(* IEC 61131-3 sources: verifaps-lib/share/PPU.stold (part 7) *)

    Pusher_states_t#PusherY1_Move_Out_White:
        {* begin(State) *}
        {* begin(onEntry) *}
        _transit := FALSE;
        {* end(onEntry) *}
        {* begin(onActive) *}
        IF ((SorterPusher1MovedOut = FALSE) AND (SorterPusher1MovedIn = TRUE)) THEN
            PusherY1 := TRUE;
        END_IF;
        {* end(onActive) *}
        {* begin(transition) *}
        IF SorterPusher1MovedOut THEN
            _transit := TRUE;
            _state := Pusher_states_t#Wait_Y1_White;
        END_IF;
        {* end(transition) *}
        {* begin(onExit) *}
        {* end(onExit) *}
        {* end(State) *}

    Pusher_states_t#PusherY2_Move_In_Black:
        {* begin(State) *}
        {* begin(onEntry) *}
        _transit := FALSE;
        {* end(onEntry) *}
        {* begin(onActive) *}
        IF ((SorterPusher2MovedOut = TRUE) AND (SorterPusher2MovedIn = FALSE)) THEN
            PusherY2 := FALSE;
        END_IF;
        {* end(onActive) *}
        {* begin(transition) *}
        IF SorterPusher2MovedIn THEN
            _transit := TRUE;
            _state := Pusher_states_t#Reset_interconnect_Slide2_Black;
        END_IF;
        {* end(transition) *}
        {* begin(onExit) *}
        {* end(onExit) *}
        {* end(State) *}

    Pusher_states_t#PusherY2_Move_In_Metal:
        {* begin(State) *}
        {* begin(onEntry) *}
        _transit := FALSE;
        {* end(onEntry) *}
        {* begin(onActive) *}
        IF ((SorterPusher2MovedOut = TRUE) AND (SorterPusher2MovedIn = FALSE)) THEN
            PusherY2 := FALSE;
        END_IF;
        {* end(onActive) *}
        {* begin(transition) *}
        IF SorterPusher2MovedIn THEN
            _transit := TRUE;
            _state := Pusher_states_t#Reset_interconnect_Slide2_Metal;
        END_IF;
        {* end(transition) *}
        {* begin(onExit) *}
        {* end(onExit) *}
        {* end(State) *}

    Pusher_states_t#PusherY2_Move_In_White:
        {* begin(State) *}
        {* begin(onEntry) *}
        _transit := FALSE;
        {* end(onEntry) *}
        {* begin(onActive) *}
        IF ((SorterPusher2MovedOut = TRUE) AND (SorterPusher2MovedIn = FALSE)) THEN
            PusherY2 := FALSE;
        END_IF;
        {* end(onActive) *}
        {* begin(transition) *}
        IF SorterPusher2MovedIn THEN
            _transit := TRUE;
            _state := Pusher_states_t#Reset_interconnect_Slide2_White;
        END_IF;
        {* end(transition) *}
        {* begin(onExit) *}
        {* end(onExit) *}
        {* end(State) *}

    Pusher_states_t#PusherY2_Move_Out_Black:
        {* begin(State) *}
        {* begin(onEntry) *}
        _transit := FALSE;
        {* end(onEntry) *}
        {* begin(onActive) *}
        IF ((SorterPusher2MovedOut = FALSE) AND (SorterPusher2MovedIn = TRUE)) THEN
            PusherY2 := TRUE;
        END_IF;
        {* end(onActive) *}
        {* begin(transition) *}
        IF SorterPusher2MovedOut THEN
            _transit := TRUE;
            _state := Pusher_states_t#Wait_Y2_Black;
        END_IF;
        {* end(transition) *}
        {* begin(onExit) *}
        {* end(onExit) *}
        {* end(State) *}

    Pusher_states_t#PusherY2_Move_Out_Metal:
        {* begin(State) *}
        {* begin(onEntry) *}
        _transit := FALSE;
        {* end(onEntry) *}
        {* begin(onActive) *}
        IF ((SorterPusher2MovedOut = FALSE) AND (SorterPusher2MovedIn = TRUE)) THEN
            PusherY2 := TRUE;
        END_IF;
        {* end(onActive) *}
        {* begin(transition) *}
        IF SorterPusher2MovedOut THEN
            _transit := TRUE;
            _state := Pusher_states_t#Wait_Y2_Metal;
        END_IF;
        {* end(transition) *}
        {* begin(onExit) *}
        {* end(onExit) *}
        {* end(State) *}

    Pusher_states_t#PusherY2_Move_Out_White:
        {* begin(State) *}
        {* begin(onEntry) *}
        _transit := FALSE;
        {* end(onEntry) *}
        {* begin(onActive) *}
        IF ((SorterPusher2MovedOut = FALSE) AND (SorterPusher2MovedIn = TRUE)) THEN
            PusherY2 := TRUE;
        END_IF;
        {* end(onActive) *}
        {* begin(transition) *}
        IF SorterPusher2MovedOut THEN
            _transit := TRUE;
            _state := Pusher_states_t#Wait_Y2_White;
        END_IF;
        {* end(transition) *}
        {* begin(onExit) *}
        {* end(onExit) *}
        {* end(State) *}

    Pusher_states_t#Reset_interconnect3:
        {* begin(State) *}
        {* begin(onEntry) *}
        _transit := FALSE;
        {* end(onEntry) *}
        {* begin(onActive) *}
        interconnect2 := FALSE;
        Timer2(IN := FALSE, PT := TIME#);
        Slide3_black := (Slide3_black - INT#1);
        Priority_Var_Black := (Priority_Var_Black - INT#1);
        {* end(onActive) *}
        {* begin(transition) *}
        IF TRUE THEN
            _transit := TRUE;
            _state := Pusher_states_t#Interstep_2;
        END_IF;
        {* end(transition) *}
        {* begin(onExit) *}
        {* end(onExit) *}
        {* end(State) *}

    Pusher_states_t#Reset_interconnect_Slide1_Black:
        {* begin(State) *}
        {* begin(onEntry) *}
        _transit := FALSE;
        {* end(onEntry) *}
        {* begin(onActive) *}
        interconnect3 := FALSE;
        Timer3(IN := FALSE, PT := TIME#);
        interconnect_Slide1_Black := FALSE;
        Timer_Slide1_Black(IN := FALSE, PT := TIME#);
        Slide1_black := (Slide1_black - INT#1);
        Priority_Var_Black := (Priority_Var_Black - INT#1);
        {* end(onActive) *}
        {* begin(transition) *}
        IF TRUE THEN
            _transit := TRUE;
            _state := Pusher_states_t#Interstep_2;
        END_IF;
        {* end(transition) *}
        {* begin(onExit) *}
        {* end(onExit) *}
        {* end(State) *}

    Pusher_states_t#Reset_interconnect_Slide1_Metal:
        {* begin(State) *}
        {* begin(onEntry) *}
        _transit := FALSE;
        {* end(onEntry) *}
        {* begin(onActive) *}
        interconnect3 := FALSE;
        Timer3(IN := FALSE, PT := TIME#);
        interconnect_Slide1_Metal := FALSE;
        Timer_Slide1_Metal(IN := FALSE, PT := TIME#);
        Slide1_metal := (Slide1_metal - INT#1);
        Priority_Var_Metal := (Priority_Var_Metal - INT#1);
        {* end(onActive) *}
        {* begin(transition) *}
        IF TRUE THEN
            _transit := TRUE;
            _state := Pusher_states_t#Interstep_2;
        END_IF;
        {* end(transition) *}
        {* begin(onExit) *}
        {* end(onExit) *}
        {* end(State) *}

    Pusher_states_t#Reset_interconnect_Slide1_White:
        {* begin(State) *}
        {* begin(onEntry) *}
        _transit := FALSE;
        {* end(onEntry) *}
        {* begin(onActive) *}
        interconnect3 := FALSE;
        Timer3(IN := FALSE, PT := TIME#);
        interconnect_Slide1_White := FALSE;
        Timer_Slide1_White(IN := FALSE, PT := TIME#);
        Slide1_white := (Slide1_white - INT#1);
        Priority_Var_White := (Priority_Var_White - INT#1);
        {* end(onActive) *}
        {* begin(transition) *}
        IF TRUE THEN
            _transit := TRUE;
            _state := Pusher_states_t#Interstep_2;
        END_IF;
        {* end(transition) *}
        {* begin(onExit) *}
        {* end(onExit) *}
        {* end(State) *}

    Pusher_states_t#Reset_interconnect_Slide2_Black:
        {* begin(State) *}
        {* begin(onEntry) *}
        _transit := FALSE;
        {* end(onEntry) *}
        {* begin(onActive) *}
        interconnect3 := FALSE;
        Timer3(IN := FALSE, PT := TIME#);
        interconnect_Slide2_Black := FALSE;
        Timer_Slide2_Black(IN := FALSE, PT := TIME#);
        Slide2_black := (Slide2_black - INT#1);
        Priority_Var_Black := (Priority_Var_Black - INT#1);
        {* end(onActive) *}
        {* begin(transition) *}
        IF TRUE THEN
            _transit := TRUE;
            _state := Pusher_states_t#Interstep_2;
        END_IF;
        {* end(transition) *}
        {* begin(onExit) *}
        {* end(onExit) *}
        {* end(State) *}

    Pusher_states_t#Reset_interconnect_Slide2_Metal:
        {* begin(State) *}
        {* begin(onEntry) *}
        _transit := FALSE;
        {* end(onEntry) *}
        {* begin(onActive) *}
        interconnect3 := FALSE;
        Timer3(IN := FALSE, PT := TIME#);
        interconnect_Slide2_Metal := FALSE;
        Timer_Slide2_Metal(IN := FALSE, PT := TIME#);
        Slide2_metal := (Slide2_metal - INT#1);
        Priority_Var_Metal := (Priority_Var_Metal - INT#1);
        {* end(onActive) *}
        {* begin(transition) *}
        IF TRUE THEN
            _transit := TRUE;
            _state := Pusher_states_t#Interstep_2;
        END_IF;
        {* end(transition) *}
        {* begin(onExit) *}
        {* end(onExit) *}
        {* end(State) *}

    Pusher_states_t#Reset_interconnect_Slide2_White:
        {* begin(State) *}
        {* begin(onEntry) *}
        _transit := FALSE;
        {* end(onEntry) *}
        {* begin(onActive) *}
        interconnect3 := FALSE;
        Timer3(IN := FALSE, PT := TIME#);
        interconnect_Slide2_White := FALSE;
        Timer_Slide2_White(IN := FALSE, PT := TIME#);
        Slide2_white := (Slide2_white - INT#1);
        Priority_Var_White := (Priority_Var_White - INT#1);
        {* end(onActive) *}
        {* begin(transition) *}
        IF TRUE THEN
            _transit := TRUE;
            _state := Pusher_states_t#Interstep_2;
        END_IF;
        {* end(transition) *}
        {* begin(onExit) *}
        {* end(onExit) *}
        {* end(State) *}

    Pusher_states_t#Reset_interconnect_Slide3_Metal:
        {* begin(State) *}
        {* begin(onEntry) *}
        _transit := FALSE;
        {* end(onEntry) *}
        {* begin(onActive) *}
        interconnect3 := FALSE;
        Timer3(IN := FALSE, PT := TIME#);
        Slide3_metal := (Slide3_metal - INT#1);
        Priority_Var_Metal := (Priority_Var_Metal - INT#1);
        {* end(onActive) *}
        {* begin(transition) *}
        IF TRUE THEN
            _transit := TRUE;
            _state := Pusher_states_t#Interstep_2;
        END_IF;
        {* end(transition) *}
        {* begin(onExit) *}
        {* end(onExit) *}
        {* end(State) *}

    Pusher_states_t#Reset_interconnect_Slide3_White:
        {* begin(State) *}
        {* begin(onEntry) *}
        _transit := FALSE;
        {* end(onEntry) *}
        {* begin(onActive) *}
        interconnect3 := FALSE;
        Timer3(IN := FALSE, PT := TIME#);
        Slide3_white := (Slide3_white - INT#1);
        Priority_Var_White := (Priority_Var_White - INT#1);
        {* end(onActive) *}
        {* begin(transition) *}
        IF TRUE THEN
            _transit := TRUE;
            _state := Pusher_states_t#Interstep_2;
        END_IF;
        {* end(transition) *}
        {* begin(onExit) *}
        {* end(onExit) *}
        {* end(State) *}

    Pusher_states_t#Second_Slide_Timer_Black:
        {* begin(State) *}
        {* begin(onEntry) *}
        _transit := FALSE;
        {* end(onEntry) *}
        {* begin(onActive) *}
        IF (SorterLightnesssensorCraneInterfaceInverse = TRUE) THEN
            Timer_Slide2_Black(IN := SorterLightnesssensorCraneInterfaceInverse, PT := Duration_Slide2_Black);
            interconnect_Slide2_Black := Timer_Slide2_Black.Q;
        END_IF;
        {* end(onActive) *}
        {* begin(transition) *}
        IF interconnect_Slide2_Black THEN
            _transit := TRUE;
            _state := Pusher_states_t#PusherY2_Move_Out_Black;
        END_IF;
        {* end(transition) *}
        {* begin(onExit) *}
        {* end(onExit) *}
        {* end(State) *}

    Pusher_states_t#Second_Slide_Timer_Metal:
        {* begin(State) *}
        {* begin(onEntry) *}
        _transit := FALSE;
        {* end(onEntry) *}
        {* begin(onActive) *}
        Timer_Slide2_Metal(IN := TRUE, PT := Duration_Slide2_Metal);
        interconnect_Slide2_Metal := Timer_Slide2_Metal.Q;
        {* end(onActive) *}
        {* begin(transition) *}
        IF interconnect_Slide2_Metal THEN
            _transit := TRUE;
            _state := Pusher_states_t#PusherY2_Move_Out_Metal;
        END_IF;
        {* end(transition) *}
        {* begin(onExit) *}
        {* end(onExit) *}
        {* end(State) *}

    Pusher_states_t#Second_Slide_Timer_White:
        {* begin(State) *}
        {* begin(onEntry) *}
        _transit := FALSE;
        {* end(onEntry) *}
        {* begin(onActive) *}
        Timer_Slide2_White(IN := TRUE, PT := Duration_Slide2_White);
        interconnect_Slide2_White := Timer_Slide2_White.Q;
        {* end(onActive) *}
        {* begin(transition) *}
        IF interconnect_Slide2_White THEN
            _transit := TRUE;
            _state := Pusher_states_t#PusherY2_Move_Out_White;
        END_IF;
        {* end(transition) *}
        {* begin(onExit) *}
        {* end(onExit) *}
        {* end(State) *}

    Pusher_states_t#Second_Slide_black_workpieces:
        {* begin(State) *}
        {* begin(onEntry) *}
        _transit := FALSE;
        {* end(onEntry) *}
        {* begin(onActive) *}
        {* end(onActive) *}
        {* begin(transition) *}
        IF TRUE THEN
            _transit := TRUE;
            _state := Pusher_states_t#Second_Slide_Timer_Black;
        END_IF;
        {* end(transition) *}
        {* begin(onExit) *}
        {* end(onExit) *}
        {* end(State) *}

    Pusher_states_t#Second_Slide_metal_workpieces:
        {* begin(State) *}
        {* begin(onEntry) *}
        _transit := FALSE;
        {* end(onEntry) *}
        {* begin(onActive) *}
        {* end(onActive) *}
        {* begin(transition) *}
        IF (SorterLightnessSensorPusher2 AND SorterCapacitiveSensorPusher2) THEN
            _transit := TRUE;
            _state := Pusher_states_t#Second_Test_For_Metal;
        END_IF;
        {* end(transition) *}
        {* begin(onExit) *}
        {* end(onExit) *}
        {* end(State) *}

    Pusher_states_t#Second_Slide_white_workpieces:
        {* begin(State) *}
        {* begin(onEntry) *}
        _transit := FALSE;
        {* end(onEntry) *}
        {* begin(onActive) *}
        {* end(onActive) *}
        {* begin(transition) *}
        IF (SorterLightnessSensorPusher2 AND NOT SorterCapacitiveSensorPusher2) THEN
            _transit := TRUE;
            _state := Pusher_states_t#Second_Test_For_White;
        END_IF;
        {* end(transition) *}
        {* begin(onExit) *}
        {* end(onExit) *}
        {* end(State) *}

    Pusher_states_t#Second_Test_For_Metal:
        {* begin(State) *}
        {* begin(onEntry) *}
        _transit := FALSE;
        {* end(onEntry) *}
        {* begin(onActive) *}
        {* end(onActive) *}
        {* begin(transition) *}
        IF TRUE THEN
            _transit := TRUE;
            _state := Pusher_states_t#Second_Slide_Timer_Metal;
        END_IF;
        {* end(transition) *}
        {* begin(onExit) *}
        {* end(onExit) *}
        {* end(State) *}

    Pusher_states_t#Second_Test_For_White:
        {* begin(State) *}
        {* begin(onEntry) *}
        _transit := FALSE;
        {* end(onEntry) *}
        {* begin(onActive) *}
        {* end(onActive) *}
        {* begin(transition) *}
        IF TRUE THEN
            _transit := TRUE;
            _state := Pusher_states_t#Second_Slide_Timer_White;
        END_IF;
        {* end(transition) *}
        {* begin(onExit) *}
        {* end(onExit) *}
        {* end(State) *}

    Pusher_states_t#Third_Slide_black_workpieces:
        {* begin(State) *}
        {* begin(onEntry) *}
        _transit := FALSE;
        {* end(onEntry) *}
        {* begin(onActive) *}
        {* end(onActive) *}
        {* begin(transition) *}
        IF (NOT SorterLightnessSensorPusher2 AND NOT SorterCapacitiveSensorPusher2) THEN
            _transit := TRUE;
            _state := Pusher_states_t#Wait_Black;
        END_IF;
        {* end(transition) *}
        {* begin(onExit) *}
        {* end(onExit) *}
        {* end(State) *}

    Pusher_states_t#Third_Slide_metal_workpieces:
        {* begin(State) *}
        {* begin(onEntry) *}
        _transit := FALSE;
        {* end(onEntry) *}
        {* begin(onActive) *}
        {* end(onActive) *}
        {* begin(transition) *}
        IF (SorterLightnessSensorPusher2 AND SorterCapacitiveSensorPusher2) THEN
            _transit := TRUE;
            _state := Pusher_states_t#Wait_Metal;
        END_IF;
        {* end(transition) *}
        {* begin(onExit) *}
        {* end(onExit) *}
        {* end(State) *}

    Pusher_states_t#Third_Slide_white_workpieces:
        {* begin(State) *}
        {* begin(onEntry) *}
        _transit := FALSE;
        {* end(onEntry) *}
        {* begin(onActive) *}
        {* end(onActive) *}
        {* begin(transition) *}
        IF (SorterLightnessSensorPusher2 AND NOT SorterCapacitiveSensorPusher2) THEN
            _transit := TRUE;
            _state := Pusher_states_t#Wait_White;
        END_IF;
        {* end(transition) *}
        {* begin(onExit) *}
        {* end(onExit) *}
        {* end(State) *}

    Pusher_states_t#Wait_Black:
        {* begin(State) *}
        {* begin(onEntry) *}
        _transit := FALSE;
        {* end(onEntry) *}
        {* begin(onActive) *}
        IF ((NOT SorterLightnessSensorPusher2 AND NOT SorterCapacitiveSensorPusher2) = TRUE) THEN
            Timer2(IN := (NOT SorterLightnessSensorPusher2 AND NOT SorterCapacitiveSensorPusher2), PT := Duration2);
            interconnect2 := Timer2.Q;
        END_IF;
        {* end(onActive) *}
        {* begin(transition) *}
        IF interconnect2 THEN
            _transit := TRUE;
            _state := Pusher_states_t#Reset_interconnect3;
        END_IF;
        {* end(transition) *}
        {* begin(onExit) *}
        {* end(onExit) *}
        {* end(State) *}

    Pusher_states_t#Wait_Metal:
        {* begin(State) *}
        {* begin(onEntry) *}
        _transit := FALSE;
        {* end(onEntry) *}
        {* begin(onActive) *}
        Timer3(IN := TRUE, PT := Duration3);
        interconnect3 := Timer3.Q;
        {* end(onActive) *}
        {* begin(transition) *}
        IF interconnect3 THEN
            _transit := TRUE;
            _state := Pusher_states_t#Reset_interconnect_Slide3_Metal;
        END_IF;
        {* end(transition) *}
        {* begin(onExit) *}
        {* end(onExit) *}
        {* end(State) *}

    Pusher_states_t#Wait_White:
        {* begin(State) *}
        {* begin(onEntry) *}
        _transit := FALSE;
        {* end(onEntry) *}
        {* begin(onActive) *}
        Timer3(IN := TRUE, PT := Duration3);
        interconnect3 := Timer3.Q;
        {* end(onActive) *}
        {* begin(transition) *}
        IF interconnect3 THEN
            _transit := TRUE;
            _state := Pusher_states_t#Reset_interconnect_Slide3_White;
        END_IF;
        {* end(transition) *}
        {* begin(onExit) *}
        {* end(onExit) *}
        {* end(State) *}

    Pusher_states_t#Wait_Y1_Black:
        {* begin(State) *}
        {* begin(onEntry) *}
        _transit := FALSE;
        {* end(onEntry) *}
        {* begin(onActive) *}
        IF (PusherY1 = TRUE) THEN
            Timer3(IN := PusherY1, PT := Duration3);
            interconnect3 := Timer3.Q;
        END_IF;
        {* end(onActive) *}
        {* begin(transition) *}
        IF interconnect3 THEN
            _transit := TRUE;
            _state := Pusher_states_t#PusherY1_Move_In_Black;
        END_IF;
        {* end(transition) *}
        {* begin(onExit) *}
        {* end(onExit) *}
        {* end(State) *}

    Pusher_states_t#Wait_Y1_Metal:
        {* begin(State) *}
        {* begin(onEntry) *}
        _transit := FALSE;
        {* end(onEntry) *}
        {* begin(onActive) *}
        IF (PusherY1 = TRUE) THEN
            Timer3(IN := PusherY1, PT := Duration3);
            interconnect3 := Timer3.Q;
        END_IF;
        {* end(onActive) *}
        {* begin(transition) *}
        IF interconnect3 THEN
            _transit := TRUE;
            _state := Pusher_states_t#PusherY1_Move_In_Metal;
        END_IF;
        {* end(transition) *}
        {* begin(onExit) *}
        {* end(onExit) *}
        {* end(State) *}

    Pusher_states_t#Wait_Y1_White:
        {* begin(State) *}
        {* begin(onEntry) *}
        _transit := FALSE;
        {* end(onEntry) *}
        {* begin(onActive) *}
        IF (PusherY1 = TRUE) THEN
            Timer3(IN := PusherY1, PT := Duration3);
            interconnect3 := Timer3.Q;
        END_IF;
        {* end(onActive) *}
        {* begin(transition) *}
        IF interconnect3 THEN
            _transit := TRUE;
            _state := Pusher_states_t#PusherY1_Move_In_White;
        END_IF;
        {* end(transition) *}
        {* begin(onExit) *}
        {* end(onExit) *}
        {* end(State) *}

    Pusher_states_t#Wait_Y2_Black:
        {* begin(State) *}
        {* begin(onEntry) *}
        _transit := FALSE;
        {* end(onEntry) *}
        {* begin(onActive) *}
        IF (PusherY2 = TRUE) THEN
            Timer3(IN := PusherY2, PT := Duration3);
            interconnect3 := Timer3.Q;
        END_IF;
        {* end(onActive) *}
        {* begin(transition) *}
        IF interconnect3 THEN
            _transit := TRUE;
            _state := Pusher_states_t#PusherY2_Move_In_Black;
        END_IF;
        {* end(transition) *}
        {* begin(onExit) *}
        {* end(onExit) *}
        {* end(State) *}

    Pusher_states_t#Wait_Y2_Metal:
        {* begin(State) *}
        {* begin(onEntry) *}
        _transit := FALSE;
        {* end(onEntry) *}
        {* begin(onActive) *}
        IF (PusherY2 = TRUE) THEN
            Timer3(IN := PusherY2, PT := Duration3);
            interconnect3 := Timer3.Q;
        END_IF;
        {* end(onActive) *}
        {* begin(transition) *}
        IF interconnect3 THEN
            _transit := TRUE;
            _state := Pusher_states_t#PusherY2_Move_In_Metal;
        END_IF;
        {* end(transition) *}
        {* begin(onExit) *}
        {* end(onExit) *}
        {* end(State) *}

    Pusher_states_t#Wait_Y2_White:
        {* begin(State) *}
        {* begin(onEntry) *}
        _transit := FALSE;
        {* end(onEntry) *}
        {* begin(onActive) *}
        IF (PusherY2 = TRUE) THEN
            Timer3(IN := PusherY2, PT := Duration3);
            interconnect3 := Timer3.Q;
        END_IF;
        {* end(onActive) *}
        {* begin(transition) *}
        IF interconnect3 THEN
            _transit := TRUE;
            _state := Pusher_states_t#PusherY2_Move_In_White;
        END_IF;
        {* end(transition) *}
        {* begin(onExit) *}
        {* end(onExit) *}
        {* end(State) *}

    END_CASE;
END_FUNCTION_BLOCK

(* ---- Scenario13_Final.xml_Conveyor.st ---- *)
FUNCTION_BLOCK Conveyor
    VAR  Duration_Conveyor_Runtime : TIME := TIME#4.0s500.0ms; END_VAR {*Lrwxp*}
    VAR  Duration_Conveyor_Test : TIME := TIME#1.0s; END_VAR {*Lrwxp*}
    VAR  SFCInit : BOOL; END_VAR {*Lrwxp*}
    VAR_INPUT  SFCReset : BOOL; END_VAR {*Irwxp*}
    VAR_OUTPUT  SorterConveyorTowardsCrane : BOOL; END_VAR {*Orwxp*}
    VAR_OUTPUT  SorterConveyorTowardsStacker : BOOL; END_VAR {*Orwxp*}
    VAR_OUTPUT  SorterGreenLampConveyor : BOOL; END_VAR {*Orwxp*}
    VAR_INPUT  SorterLightbarrierCraneInterface : BOOL; END_VAR {*Irwxp*}
    VAR_INPUT  SorterStartButton : BOOL; END_VAR {*Irwxp*}
    VAR_INPUT  SorterSwitchManuellAutomatic : BOOL; END_VAR {*Irwxp*}
    VAR_OUTPUT  SorterWhiteLampConveyor : BOOL; END_VAR {*Orwxp*}
    VAR_OUTPUT  StartCommandConveyor : BOOL; END_VAR {*Orwxp*}
    VAR_INPUT  StartVar : BOOL; END_VAR {*Irwxp*}
    VAR  Timer_Conveyor_Runtime : TON; END_VAR {*Lrwxp*}
    VAR  Timer_Conveyor_Test : TON; END_VAR {*Lrwxp*}
    VAR  _state : Conveyor_states_t; END_VAR {*Lrwxp*}
    VAR  _transit : BOOL; END_VAR {*Lrwxp*}
    VAR  interconnectConveyorStartCommand : BOOL; END_VAR {*Lrwxp*}
    VAR  interconnectConveyorTerminationCommand : BOOL; END_VAR {*Lrwxp*}
    VAR  interconnect_Conveyor_Runtime : BOOL; END_VAR {*Lrwxp*}
    VAR  interconnect_Conveyor_Test : BOOL; END_VAR {*Lrwxp*}

    CASE _state OF
        Conveyor_states_t#Conveyor_Init:
            {* begin(State) *}
            {* begin(onEntry) *}
            _transit := FALSE;
            {* end(onEntry) *}
            {* begin(onActive) *}
            SorterConveyorTowardsStacker := TRUE;
            SorterConveyorTowardsCrane := FALSE;
            Timer_Conveyor_Test(IN := TRUE, PT := Duration_Conveyor_Test);
            interconnect_Conveyor_Test := Timer_Conveyor_Test.Q;
            {* end(onActive) *}
            {* begin(transition) *}
            IF interconnect_Conveyor_Test THEN
                _transit := TRUE;
                _state := Conveyor_states_t#Conveyor_init_2;
            END_IF;
            {* end(transition) *}
            {* begin(onExit) *}
            {* end(onExit) *}
            {* end(State) *}

        Conveyor_states_t#Conveyor_Stop_Empty_Magazin:
            {* begin(State) *}
            {* begin(onEntry) *}
            _transit := FALSE;
            {* end(onEntry) *}
            {* begin(onActive) *}
            SorterConveyorTowardsStacker := FALSE;
            SorterConveyorTowardsCrane := FALSE;
            interconnectConveyorStartCommand := FALSE;
            {* end(onActive) *}
            {* begin(transition) *}
            IF TRUE THEN
                _transit := TRUE;
                _state := Conveyor_states_t#Interstep;
            END_IF;
            {* end(transition) *}
            {* begin(onExit) *}
            {* end(onExit) *}
            {* end(State) *}

        Conveyor_states_t#Conveyor_Towards_Stacker:
            {* begin(State) *}
            {* begin(onEntry) *}
            _transit := FALSE;
            {* end(onEntry) *}
            {* begin(onActive) *}
            SorterConveyorTowardsStacker := TRUE;
            SorterConveyorTowardsCrane := FALSE;
            {* end(onActive) *}
            {* begin(transition) *}
            IF TRUE THEN
                _transit := TRUE;
                _state := Conveyor_states_t#Runtime_Conveyor;
            END_IF;
            {* end(transition) *}
            {* begin(onExit) *}
            {* end(onExit) *}
            {* end(State) *}

        Conveyor_states_t#Conveyor_init_2:
            {* begin(State) *}
            {* begin(onEntry) *}
            _transit := FALSE;
            {* end(onEntry) *}
            {* begin(onActive) *}
            SorterConveyorTowardsStacker := FALSE;
            SorterConveyorTowardsCrane := FALSE;
            interconnect_Conveyor_Test := FALSE;
            Timer_Conveyor_Test(IN := FALSE, PT := TIME#);
            {* end(onActive) *}
            {* begin(transition) *}
            IF TRUE THEN
                _transit := TRUE;
                _state := Conveyor_states_t#Interstep;
            END_IF;
            {* end(transition) *}
            {* begin(onExit) *}
            {* end(onExit) *}
            {* end(State) *}

        Conveyor_states_t#Conveyor_pause:
            {* begin(State) *}
            {* begin(onEntry) *}
            _transit := FALSE;
            {* end(onEntry) *}
            {* begin(onActive) *}
            SorterConveyorTowardsStacker := FALSE;
            SorterConveyorTowardsCrane := FALSE;
            interconnect_Conveyor_Runtime := FALSE;
            Timer_Conveyor_Runtime(IN := FALSE, PT := TIME#);
            {* end(onActive) *}
            {* begin(transition) *}
            IF TRUE THEN
                _transit := TRUE;
                _state := Conveyor_states_t#Interstep;
            END_IF;
            {* end(transition) *}
            {* begin(onExit) *}
            {* end(onExit) *}
            {* end(State) *}

        Conveyor_states_t#Green_Lamp:
            {* begin(State) *}
            {* begin(onEntry) *}
            _transit := FALSE;
            {* end(onEntry) *}
            {* begin(onActive) *}
            SorterGreenLampConveyor := TRUE;
            interconnectConveyorStartCommand := FALSE;
            {* end(onActive) *}
            {* begin(transition) *}
            IF TRUE THEN
                _transit := TRUE;
                _state := Conveyor_states_t#Conveyor_Init;
            END_IF;
            {* end(transition) *}
            {* begin(onExit) *}
            {* end(onExit) *}
            {* end(State) *}

        Conveyor_states_t#Init:
            {* begin(State) *}
            {* begin(onEntry) *}
            _transit := FALSE;
            {* end(onEntry) *}
            {* begin(onActive) *}
            {* end(onActive) *}
            {* begin(transition) *}
            IF TRUE THEN
                _transit := TRUE;
                _state := Conveyor_states_t#Start_Conveyor;
            END_IF;
            {* end(transition) *}
            {* begin(onExit) *}
            {* end(onExit) *}
            {* end(State) *}

        Conveyor_states_t#Interstep:
            {* begin(State) *}
            {* begin(onEntry) *}
            _transit := FALSE;
            {* end(onEntry) *}
            {* begin(onActive) *}
            StartCommandConveyor := TRUE;
            {* end(onActive) *}
            {* begin(transition) *}
            IF StartVar THEN
                _transit := TRUE;
                _state := Conveyor_states_t#Step0;
            END_IF;
            {* end(transition) *}
            {* begin(onExit) *}
            {* end(onExit) *}
            {* end(State) *}

        Conveyor_states_t#Runtime_Conveyor:
            {* begin(State) *}
            {* begin(onEntry) *}
            _transit := FALSE;
            {* end(onEntry) *}
            {* begin(onActive) *}
            Timer_Conveyor_Runtime(IN := TRUE, PT := Duration_Conveyor_Runtime);
            interconnect_Conveyor_Runtime := Timer_Conveyor_Runtime.Q;
            {* end(onActive) *}
            {* begin(transition) *}
            IF interconnect_Conveyor_Runtime THEN
                _transit := TRUE;
                _state := Conveyor_states_t#Conveyor_pause;
            END_IF;
            {* end(transition) *}
            {* begin(onExit) *}
            {* end(onExit) *}
            {* end(State) *}

        Conveyor_states_t#Start_Conveyor:
            {* begin(State) *}
            {* begin(onEntry) *}
            _transit := FALSE;
            {* end(onEntry) *}
            {* begin(onActive) *}
            interconnectConveyorTerminationCommand := FALSE;
            SorterConveyorTowardsStacker := FALSE;
            SorterConveyorTowardsCrane := FALSE;
            SorterGreenLampConveyor := FALSE;
            interconnect_Conveyor_Runtime := FALSE;
            interconnect_Conveyor_Test := FALSE;
            Timer_Conveyor_Test(IN := FALSE, PT := TIME#);
            Timer_Conveyor_Runtime(IN := FALSE, PT := TIME#);
            StartVar := FALSE;
            StartCommandConveyor := FALSE;
            IF (SorterStartButton = TRUE) THEN
                interconnectConveyorStartCommand := TRUE;
            END_IF;
            {* end(onActive) *}
            {* begin(transition) *}
            IF interconnectConveyorStartCommand THEN
                _transit := TRUE;
                _state := Conveyor_states_t#Green_Lamp;
            END_IF;
            {* end(transition) *}
            {* begin(onExit) *}
            {* end(onExit) *}
            {* end(State) *}

        Conveyor_states_t#Step0:
            {* begin(State) *}
            {* begin(onEntry) *}
            _transit := FALSE;
            {* end(onEntry) *}
            {* begin(onActive) *}
            {* end(onActive) *}
            {* begin(transition) *}
            IF SorterLightbarrierCraneInterface THEN
                _transit := TRUE;
                _state := Conveyor_states_t#Conveyor_Towards_Stacker;
            ELSEIF NOT SorterLightbarrierCraneInterface THEN
                _transit := TRUE;
                _state := Conveyor_states_t#Conveyor_Stop_Empty_Magazin;
            END_IF;
            {* end(transition) *}
            {* begin(onExit) *}
            {* end(onExit) *}
            {* end(State) *}

            END_CASE;
END_FUNCTION_BLOCK

(* ---- Scenario13_Final.xml_Crane.st ---- *)
FUNCTION_BLOCK Crane
    VAR_INPUT  AnalogCranePosition : INT; END_VAR {*Irwxp*}
    VAR_OUTPUT  AnalogCranePressure : INT; END_VAR {*Orwxp*}
    VAR_INPUT  CraneDown : BOOL; END_VAR {*Irwxp*}
    VAR_OUTPUT  CraneLower : BOOL; END_VAR {*Orwxp*}
    VAR_INPUT  CraneSucked : BOOL; END_VAR {*Irwxp*}
    VAR_OUTPUT  CraneTurnClockwise : BOOL; END_VAR {*Orwxp*}
    VAR_OUTPUT  CraneTurnCounterclockwise : BOOL; END_VAR {*Orwxp*}
    VAR_INPUT  CraneUp : BOOL; END_VAR {*Irwxp*}
    VAR  Duration1 : TIME := TIME#1.0s500.0ms; END_VAR {*Lrwxp*}
    VAR_INPUT  MagazinCapacitiveSensor : BOOL; END_VAR {*Irwxp*}
    VAR_INPUT  MagazinOpticalSensor : BOOL; END_VAR {*Irwxp*}
    VAR_OUTPUT  MagazinSlider : BOOL; END_VAR {*Orwxp*}
    VAR_OUTPUT  MagazinVacuumOff : BOOL; END_VAR {*Orwxp*}
    VAR_OUTPUT  MagazinVacuumOn : BOOL; END_VAR {*Orwxp*}
    VAR  SFCInit : BOOL; END_VAR {*Lrwxp*}
    VAR_INPUT  SFCReset : BOOL; END_VAR {*Irwxp*}
    VAR_INPUT  SliderMovedOut : BOOL; END_VAR {*Irwxp*}
    VAR_INPUT  SliderNotMovedOut : BOOL; END_VAR {*Irwxp*}
    VAR_INPUT  StampLowered : BOOL; END_VAR {*Irwxp*}
    VAR_INPUT  StampSliderFilled : BOOL; END_VAR {*Irwxp*}
    VAR_INPUT  StampSliderSensorMovedOut : BOOL; END_VAR {*Irwxp*}
    VAR_INPUT  StartButtonMagazin : BOOL; END_VAR {*Irwxp*}
    VAR_OUTPUT  StartCommandCrane : BOOL; END_VAR {*Orwxp*}
    VAR_INPUT  StartVar : BOOL; END_VAR {*Irwxp*}
    VAR  TimeDelay_Timer : TON; END_VAR {*Lrwxp*}
    VAR  TimeDelay_Timer_Duration : TIME := TIME#50.0ms; END_VAR {*Lrwxp*}
    VAR  TimeDelay_Timer_interconnect : BOOL; END_VAR {*Lrwxp*}
    VAR  Timer1 : TON; END_VAR {*Lrwxp*}
    VAR_INPUT  WorkpieceReady : BOOL; END_VAR {*Irwxp*}
    VAR  _state : Crane_states_t; END_VAR {*Lrwxp*}
    VAR  _transit : BOOL; END_VAR {*Lrwxp*}
    VAR  actualtime1 : TIME; END_VAR {*Lrwxp*}
    VAR  interconnect : BOOL; END_VAR {*Lrwxp*}
    VAR  interconnectCraneStartCommand : BOOL; END_VAR {*Lrwxp*}

    CASE _state OF
        Crane_states_t#Crane_Go_Up:
            {* begin(State) *}
            {* begin(onEntry) *}
            _transit := FALSE;
            {* end(onEntry) *}
            {* begin(onActive) *}
            CraneLower := FALSE;
            {* end(onActive) *}
            {* begin(transition) *}
            IF CraneUp THEN
                _transit := TRUE;
                _state := Crane_states_t#Step3;
            END_IF;
            {* end(transition) *}
            {* begin(onExit) *}
            {* end(onExit) *}
            {* end(State) *}

        Crane_states_t#Crane_Go_Up_White:
            {* begin(State) *}
            {* begin(onEntry) *}
            _transit := FALSE;
            {* end(onEntry) *}
            {* begin(onActive) *}
            CraneLower := FALSE;
            {* end(onActive) *}
            {* begin(transition) *}
            IF CraneUp THEN
                _transit := TRUE;
                _state := Crane_states_t#Step3;
            END_IF;
            {* end(transition) *}
            {* begin(onExit) *}
            {* end(onExit) *}
            {* end(State) *}

        Crane_states_t#Crane_Init:
            {* begin(State) *}
            {* begin(onEntry) *}
            _transit := FALSE;
            {* end(onEntry) *}
            {* begin(onActive) *}
            CraneLower := TRUE;
            interconnectCraneStartCommand := FALSE;
            AnalogCranePressure := INT#6000;
            {* end(onActive) *}
            {* begin(transition) *}
            IF CraneDown THEN
                _transit := TRUE;
                _state := Crane_states_t#Crane_Init_2;
            END_IF;
            {* end(transition) *}
            {* begin(onExit) *}
            {* end(onExit) *}
            {* end(State) *}

        Crane_states_t#Crane_Init_2:
            {* begin(State) *}
            {* begin(onEntry) *}
            _transit := FALSE;
            {* end(onEntry) *}
            {* begin(onActive) *}
            CraneLower := FALSE;
            {* end(onActive) *}
            {* begin(transition) *}
            IF CraneUp THEN
                _transit := TRUE;
                _state := Crane_states_t#Interstep;
            END_IF;
            {* end(transition) *}
            {* begin(onExit) *}
            {* end(onExit) *}
            {* end(State) *}

        Crane_states_t#Crane_Lift_At_Stamp:
            {* begin(State) *}
            {* begin(onEntry) *}
            _transit := FALSE;
            {* end(onEntry) *}
            {* begin(onActive) *}
            CraneLower := FALSE;
            {* end(onActive) *}
            {* begin(transition) *}
            IF CraneUp THEN
                _transit := TRUE;
                _state := Crane_states_t#Crane_Turn_Left_From_Stamp;
            END_IF;
            {* end(transition) *}
            {* begin(onExit) *}
            {* end(onExit) *}
            {* end(State) *}

        Crane_states_t#Crane_Lift_At_Stamp2:
            {* begin(State) *}
            {* begin(onEntry) *}
            _transit := FALSE;
            {* end(onEntry) *}
            {* begin(onActive) *}
            CraneLower := FALSE;
            AnalogCranePressure := INT#0;
            {* end(onActive) *}
            {* begin(transition) *}
            IF CraneUp THEN
                _transit := TRUE;
                _state := Crane_states_t#Crane_Turn_Right_From_Stamp;
            END_IF;
            {* end(transition) *}
            {* begin(onExit) *}
            {* end(onExit) *}
            {* end(State) *}

        Crane_states_t#Crane_Lift_Conveyor:
            {* begin(State) *}
            {* begin(onEntry) *}
            _transit := FALSE;
            {* end(onEntry) *}
            {* begin(onActive) *}
            CraneLower := FALSE;
            {* end(onActive) *}
            {* begin(transition) *}
            IF TRUE THEN
                _transit := TRUE;
                _state := Crane_states_t#Interstep;
            END_IF;
            {* end(transition) *}
            {* begin(onExit) *}
            {* end(onExit) *}
            {* end(State) *}

        Crane_states_t#Crane_Lift_Conveyor2:
            {* begin(State) *}
            {* begin(onEntry) *}
            _transit := FALSE;
            {* end(onEntry) *}
            {* begin(onActive) *}
            CraneLower := FALSE;
            {* end(onActive) *}
            {* begin(transition) *}
            IF TRUE THEN
                _transit := TRUE;
                _state := Crane_states_t#Interstep;
            END_IF;
            {* end(transition) *}
            {* begin(onExit) *}
            {* end(onExit) *}
            {* end(State) *}

        Crane_states_t#Crane_Lift_Conveyor_Black:
            {* begin(State) *}
            {* begin(onEntry) *}
            _transit := FALSE;
            {* end(onEntry) *}
            {* begin(onActive) *}
            CraneLower := FALSE;
            {* end(onActive) *}
            {* begin(transition) *}
            IF CraneUp THEN
                _transit := TRUE;
                _state := Crane_states_t#Crane_Turn_Left_Back_To_Stamp;
            END_IF;
            {* end(transition) *}
            {* begin(onExit) *}
            {* end(onExit) *}
            {* end(State) *}

        Crane_states_t#Crane_Lift_Magazin:
            {* begin(State) *}
            {* begin(onEntry) *}
            _transit := FALSE;
            {* end(onEntry) *}
            {* begin(onActive) *}
            CraneLower := FALSE;
            {* end(onActive) *}
            {* begin(transition) *}
            IF CraneUp THEN
                _transit := TRUE;
                _state := Crane_states_t#Crane_Turn_Left_NOT_Metallic;
            END_IF;
            {* end(transition) *}
            {* begin(onExit) *}
            {* end(onExit) *}
            {* end(State) *}

        Crane_states_t#Crane_Lift_Magazin_Metallic:
            {* begin(State) *}
            {* begin(onEntry) *}
            _transit := FALSE;
            {* end(onEntry) *}
            {* begin(onActive) *}
            CraneLower := FALSE;
            {* end(onActive) *}
            {* begin(transition) *}
            IF CraneUp THEN
                _transit := TRUE;
                _state := Crane_states_t#Crane_Turn_Left_Metallic;
            END_IF;
            {* end(transition) *}
            {* begin(onExit) *}
            {* end(onExit) *}
            {* end(State) *}

        Crane_states_t#Crane_Lift_Magazin_White:
            {* begin(State) *}
            {* begin(onEntry) *}
            _transit := FALSE;
            {* end(onEntry) *}
            {* begin(onActive) *}
            CraneLower := FALSE;
            {* end(onActive) *}
            {* begin(transition) *}
            IF CraneUp THEN
                _transit := TRUE;
                _state := Crane_states_t#Crane_Turn_Left_White;
            END_IF;
            {* end(transition) *}
            {* begin(onExit) *}
            {* end(onExit) *}
            {* end(State) *}

        Crane_states_t#Crane_Lift_NOT_Metallic_Black:
            {* begin(State) *}
            {* begin(onEntry) *}
            _transit := FALSE;
            {* end(onEntry) *}
            {* begin(onActive) *}
            CraneLower := FALSE;
            {* end(onActive) *}
            {* begin(transition) *}
            IF CraneUp THEN
                _transit := TRUE;
                _state := Crane_states_t#Crane_Turn_Left_NOT_Metallic_Black;
            END_IF;
            {* end(transition) *}
            {* begin(onExit) *}
            {* end(onExit) *}
            {* end(State) *}

        Crane_states_t#Crane_Lower:
            {* begin(State) *}
            {* begin(onEntry) *}
            _transit := FALSE;
            {* end(onEntry) *}
            {* begin(onActive) *}
            MagazinVacuumOn := TRUE;
            MagazinVacuumOff := FALSE;
            CraneLower := TRUE;
            AnalogCranePressure := INT#0;
            {* end(onActive) *}
            {* begin(transition) *}
            IF CraneSucked THEN
                _transit := TRUE;
                _state := Crane_states_t#Step0;
            END_IF;
            {* end(transition) *}
            {* begin(onExit) *}
            {* end(onExit) *}
            {* end(State) *}

        Crane_states_t#Crane_On_Conveyor:
            {* begin(State) *}
            {* begin(onEntry) *}
            _transit := FALSE;
            {* end(onEntry) *}
            {* begin(onActive) *}
            CraneTurnCounterclockwise := FALSE;
            CraneTurnClockwise := FALSE;
            CraneLower := TRUE;
            {* end(onActive) *}
            {* begin(transition) *}
            IF CraneDown THEN
                _transit := TRUE;
                _state := Crane_states_t#release;
            END_IF;
            {* end(transition) *}
            {* begin(onExit) *}
            {* end(onExit) *}
            {* end(State) *}

        Crane_states_t#Crane_On_Conveyor_Metallic:
            {* begin(State) *}
            {* begin(onEntry) *}
            _transit := FALSE;
            {* end(onEntry) *}
            {* begin(onActive) *}
            CraneTurnCounterclockwise := FALSE;
            CraneTurnClockwise := FALSE;
            CraneLower := TRUE;
            {* end(onActive) *}
            {* begin(transition) *}
            IF CraneDown THEN
                _transit := TRUE;
                _state := Crane_states_t#release;
            END_IF;
            {* end(transition) *}
            {* begin(onExit) *}
            {* end(onExit) *}
            {* end(State) *}

        Crane_states_t#Crane_On_Conveyor_Metallic2:
            {* begin(State) *}
            {* begin(onEntry) *}
            _transit := FALSE;
            {* end(onEntry) *}
            {* begin(onActive) *}
            CraneTurnCounterclockwise := FALSE;
            CraneTurnClockwise := FALSE;
            CraneLower := TRUE;
            {* end(onActive) *}
            {* begin(transition) *}
            IF CraneDown THEN
                _transit := TRUE;
                _state := Crane_states_t#release2;
            END_IF;
            {* end(transition) *}
            {* begin(onExit) *}
            {* end(onExit) *}
            {* end(State) *}

        Crane_states_t#Crane_On_Conveyor_Not_Metallica_Black:
            {* begin(State) *}
            {* begin(onEntry) *}
            _transit := FALSE;
            {* end(onEntry) *}
            {* begin(onActive) *}
            CraneTurnCounterclockwise := FALSE;
            CraneTurnClockwise := FALSE;
            CraneLower := TRUE;
            {* end(onActive) *}
            {* begin(transition) *}
            IF CraneDown THEN
                _transit := TRUE;
                _state := Crane_states_t#release_Black;
            END_IF;
            {* end(transition) *}
            {* begin(onExit) *}
            {* end(onExit) *}
            {* end(State) *}

        Crane_states_t#Crane_On_Stamp_Metallic:
            {* begin(State) *}
            {* begin(onEntry) *}
            _transit := FALSE;
            {* end(onEntry) *}
            {* begin(onActive) *}
            CraneTurnCounterclockwise := FALSE;
            CraneTurnClockwise := FALSE;
            CraneLower := TRUE;
            {* end(onActive) *}
            {* begin(transition) *}
            IF CraneDown THEN
                _transit := TRUE;
                _state := Crane_states_t#release_Workpiece;
            END_IF;
            {* end(transition) *}
            {* begin(onExit) *}
            {* end(onExit) *}
            {* end(State) *}

        Crane_states_t#Crane_On_Stamp_Metallic2:
            {* begin(State) *}
            {* begin(onEntry) *}
            _transit := FALSE;
            {* end(onEntry) *}
            {* begin(onActive) *}
            CraneTurnCounterclockwise := FALSE;
            CraneTurnClockwise := FALSE;
            {* end(onActive) *}
            {* begin(transition) *}
            IF StampLowered THEN
                _transit := TRUE;
                _state := Crane_states_t#Interstep_4;
            END_IF;
            {* end(transition) *}
            {* begin(onExit) *}
            {* end(onExit) *}
            {* end(State) *}

        Crane_states_t#Crane_On_Stamp_Metallic2_Lower:
            {* begin(State) *}
            {* begin(onEntry) *}
            _transit := FALSE;
            {* end(onEntry) *}
            {* begin(onActive) *}
            CraneLower := TRUE;
            {* end(onActive) *}
            {* begin(transition) *}
            IF CraneDown THEN
                _transit := TRUE;
                _state := Crane_states_t#Suck_At_Stamp2;
            END_IF;
            {* end(transition) *}
            {* begin(onExit) *}
            {* end(onExit) *}
            {* end(State) *}

        Crane_states_t#Crane_On_Stamp_Stop_Black:
            {* begin(State) *}
            {* begin(onEntry) *}
            _transit := FALSE;
            {* end(onEntry) *}
            {* begin(onActive) *}
            CraneTurnClockwise := FALSE;
            CraneTurnCounterclockwise := FALSE;
            {* end(onActive) *}
            {* begin(transition) *}
            IF TRUE THEN
                _transit := TRUE;
                _state := Crane_states_t#Reset_interconnect;
            END_IF;
            {* end(transition) *}
            {* begin(onExit) *}
            {* end(onExit) *}
            {* end(State) *}

        Crane_states_t#Crane_On_Stamp_White:
            {* begin(State) *}
            {* begin(onEntry) *}
            _transit := FALSE;
            {* end(onEntry) *}
            {* begin(onActive) *}
            CraneTurnCounterclockwise := FALSE;
            CraneTurnClockwise := FALSE;
            CraneLower := TRUE;
            {* end(onActive) *}
            {* begin(transition) *}
            IF CraneDown THEN
                _transit := TRUE;
                _state := Crane_states_t#release_Workpiece_White;
            END_IF;
            {* end(transition) *}
            {* begin(onExit) *}
            {* end(onExit) *}
            {* end(State) *}

        Crane_states_t#Crane_Turn_Left_Back_To_Stamp:
            {* begin(State) *}
            {* begin(onEntry) *}
            _transit := FALSE;
            {* end(onEntry) *}
            {* begin(onActive) *}
            CraneTurnCounterclockwise := TRUE;
            CraneTurnClockwise := FALSE;
            {* end(onActive) *}
            {* begin(transition) *}
            IF ((AnalogCranePosition > INT#8160) AND (AnalogCranePosition < INT#8260)) THEN
                _transit := TRUE;
                _state := Crane_states_t#Crane_On_Stamp_Stop_Black;
            END_IF;
            {* end(transition) *}
            {* begin(onExit) *}
            {* end(onExit) *}
            {* end(State) *}

        Crane_states_t#Crane_Turn_Left_From_Stamp:
            {* begin(State) *}
            {* begin(onEntry) *}
            _transit := FALSE;
            {* end(onEntry) *}
            {* begin(onActive) *}
            CraneTurnClockwise := TRUE;
            CraneTurnCounterclockwise := FALSE;
            {* end(onActive) *}
            {* begin(transition) *}
            IF ((AnalogCranePosition > INT#16060) AND (AnalogCranePosition < INT#16160)) THEN
                _transit := TRUE;
                _state := Crane_states_t#Crane_On_Conveyor_Metallic;
            END_IF;
            {* end(transition) *}
            {* begin(onExit) *}
            {* end(onExit) *}
            {* end(State) *}

        Crane_states_t#Crane_Turn_Left_Metallic:
            {* begin(State) *}
            {* begin(onEntry) *}
            _transit := FALSE;
            {* end(onEntry) *}
            {* begin(onActive) *}
            CraneTurnCounterclockwise := TRUE;
            CraneTurnClockwise := FALSE;
            {* end(onActive) *}
            {* begin(transition) *}
            IF ((AnalogCranePosition > INT#8160) AND (AnalogCranePosition < INT#8260)) THEN
                _transit := TRUE;
                _state := Crane_states_t#Crane_On_Stamp_Metallic;
            END_IF;
            {* end(transition) *}
            {* begin(onExit) *}
            {* end(onExit) *}
            {* end(State) *}

        Crane_states_t#Crane_Turn_Left_Metallic2:
            {* begin(State) *}
            {* begin(onEntry) *}
            _transit := FALSE;
            {* end(onEntry) *}
            {* begin(onActive) *}
            CraneTurnCounterclockwise := TRUE;
            CraneTurnClockwise := FALSE;
            {* end(onActive) *}
            {* begin(transition) *}
            IF ((AnalogCranePosition > INT#8160) AND (AnalogCranePosition < INT#8260)) THEN
                _transit := TRUE;
                _state := Crane_states_t#Crane_On_Stamp_Metallic2;
            END_IF;
            {* end(transition) *}
            {* begin(onExit) *}
            {* end(onExit) *}
            {* end(State) *}

        Crane_states_t#Crane_Turn_Left_NOT_Metallic:
            {* begin(State) *}
            {* begin(onEntry) *}
            _transit := FALSE;
            {* end(onEntry) *}
            {* begin(onActive) *}
            CraneTurnCounterclockwise := TRUE;
            CraneTurnClockwise := FALSE;
            {* end(onActive) *}
            {* begin(transition) *}
            IF ((AnalogCranePosition > INT#16160) AND (AnalogCranePosition < INT#16260)) THEN
                _transit := TRUE;
                _state := Crane_states_t#Crane_On_Conveyor;
            END_IF;
            {* end(transition) *}
            {* begin(onExit) *}
            {* end(onExit) *}
            {* end(State) *}

        Crane_states_t#Crane_Turn_Left_NOT_Metallic_Black:
            {* begin(State) *}
            {* begin(onEntry) *}
            _transit := FALSE;
            {* end(onEntry) *}
            {* begin(onActive) *}
            CraneTurnCounterclockwise := TRUE;
            CraneTurnClockwise := FALSE;
            {* end(onActive) *}
            {* begin(transition) *}
            IF ((AnalogCranePosition > INT#16160) AND (AnalogCranePosition < INT#16260)) THEN
                _transit := TRUE;
                _state := Crane_states_t#Crane_On_Conveyor_Not_Metallica_Black;
            END_IF;
            {* end(transition) *}
            {* begin(onExit) *}
            {* end(onExit) *}
            {* end(State) *}

        Crane_states_t#Crane_Turn_Left_White:
            {* begin(State) *}
            {* begin(onEntry) *}
            _transit := FALSE;
            {* end(onEntry) *}
            {* begin(onActive) *}
            CraneTurnCounterclockwise := TRUE;
            CraneTurnClockwise := FALSE;
            {* end(onActive) *}
            {* begin(transition) *}
            IF ((AnalogCranePosition > INT#8160) AND (AnalogCranePosition < INT#8260)) THEN
                _transit := TRUE;
                _state := Crane_states_t#Crane_On_Stamp_White;
            END_IF;
            {* end(transition) *}
            {* begin(onExit) *}
            {* end(onExit) *}
            {* end(State) *}

        Crane_states_t#Crane_Turn_Right_From_Stamp:
            {* begin(State) *}
            {* begin(onEntry) *}
            _transit := FALSE;
            {* end(onEntry) *}
            {* begin(onActive) *}
            CraneTurnClockwise := TRUE;
            CraneTurnCounterclockwise := FALSE;
            {* end(onActive) *}
            {* begin(transition) *}
            IF ((AnalogCranePosition > INT#16160) AND (AnalogCranePosition < INT#16260)) THEN
                _transit := TRUE;
                _state := Crane_states_t#Crane_On_Conveyor_Metallic2;
            END_IF;
            {* end(transition) *}
            {* begin(onExit) *}
            {* end(onExit) *}
            {* end(State) *}

        Crane_states_t#Init:
            {* begin(State) *}
            {* begin(onEntry) *}
            _transit := FALSE;
            {* end(onEntry) *}
            {* begin(onActive) *}
            {* end(onActive) *}
            {* begin(transition) *}
            IF TRUE THEN
                _transit := TRUE;
                _state := Crane_states_t#Start_Crane;
            END_IF;
            {* end(transition) *}
            {* begin(onExit) *}
            {* end(onExit) *}
            {* end(State) *}

        Crane_states_t#Interstep:
            {* begin(State) *}
            {* begin(onEntry) *}
            _transit := FALSE;
            {* end(onEntry) *}
            {* begin(onActive) *}
            StartCommandCrane := TRUE;
            {* end(onActive) *}
            {* begin(transition) *}
            IF StartVar THEN
                _transit := TRUE;
                _state := Crane_states_t#Interstep_2;
            END_IF;
            {* end(transition) *}
            {* begin(onExit) *}
            {* end(onExit) *}
            {* end(State) *}

        Crane_states_t#Interstep_2:
            {* begin(State) *}
            {* begin(onEntry) *}
            _transit := FALSE;
            {* end(onEntry) *}
            {* begin(onActive) *}
            {* end(onActive) *}
            {* begin(transition) *}
            IF SliderMovedOut THEN
                _transit := TRUE;
                _state := Crane_states_t#TimeDelay;
            END_IF;
            {* end(transition) *}
            {* begin(onExit) *}
            {* end(onExit) *}
            {* end(State) *}

        Crane_states_t#Interstep_3:
            {* begin(State) *}
            {* begin(onEntry) *}
            _transit := FALSE;
            {* end(onEntry) *}
            {* begin(onActive) *}
            {* end(onActive) *}
            {* begin(transition) *}
            IF NOT WorkpieceReady THEN
                _transit := TRUE;
                _state := Crane_states_t#No_Workpiece_ready;
            ELSEIF WorkpieceReady THEN
                _transit := TRUE;
                _state := Crane_states_t#Turn_Right;
            END_IF;
            {* end(transition) *}
            {* begin(onExit) *}
            {* end(onExit) *}
            {* end(State) *}

        Crane_states_t#Interstep_4:
            {* begin(State) *}
            {* begin(onEntry) *}
            _transit := FALSE;
            {* end(onEntry) *}
            {* begin(onActive) *}
            {* end(onActive) *}
            {* begin(transition) *}
            IF StampSliderSensorMovedOut THEN
                _transit := TRUE;
                _state := Crane_states_t#Crane_On_Stamp_Metallic2_Lower;
            END_IF;
            {* end(transition) *}
            {* begin(onExit) *}
            {* end(onExit) *}
            {* end(State) *}

        Crane_states_t#Lower_Crane:
            {* begin(State) *}
            {* begin(onEntry) *}
            _transit := FALSE;
            {* end(onEntry) *}
            {* begin(onActive) *}
            CraneLower := TRUE;
            {* end(onActive) *}
            {* begin(transition) *}
            IF CraneDown THEN
                _transit := TRUE;
                _state := Crane_states_t#Suck_At_Stamp;
            END_IF;
            {* end(transition) *}
            {* begin(onExit) *}
            {* end(onExit) *}
            {* end(State) *}

        Crane_states_t#Magazin_Stop:
            {* begin(State) *}
            {* begin(onEntry) *}
            _transit := FALSE;
            {* end(onEntry) *}
            {* begin(onActive) *}
            CraneTurnClockwise := FALSE;
            CraneTurnCounterclockwise := FALSE;
            {* end(onActive) *}
            {* begin(transition) *}
            IF TRUE THEN
                _transit := TRUE;
                _state := Crane_states_t#Crane_Lower;
            END_IF;
            {* end(transition) *}
            {* begin(onExit) *}
            {* end(onExit) *}
            {* end(State) *}

        Crane_states_t#Magazin_Stop_Black:
            {* begin(State) *}
            {* begin(onEntry) *}
            _transit := FALSE;
            {* end(onEntry) *}
            {* begin(onActive) *}
            CraneTurnClockwise := FALSE;
            CraneTurnCounterclockwise := FALSE;
            MagazinVacuumOn := TRUE;
            MagazinVacuumOff := FALSE;
            CraneLower := TRUE;
            {* end(onActive) *}
            {* begin(transition) *}
            IF CraneSucked THEN
                _transit := TRUE;
                _state := Crane_states_t#Crane_Lift_NOT_Metallic_Black;
            END_IF;
            {* end(transition) *}
            {* begin(onExit) *}
            {* end(onExit) *}
            {* end(State) *}

        Crane_states_t#Magazin_Stop_Final:
            {* begin(State) *}
            {* begin(onEntry) *}
            _transit := FALSE;
            {* end(onEntry) *}
            {* begin(onActive) *}
            CraneTurnClockwise := FALSE;
            CraneTurnCounterclockwise := FALSE;
            {* end(onActive) *}
            {* begin(transition) *}
            IF TRUE THEN
                _transit := TRUE;
                _state := Crane_states_t#Start_Crane;
            END_IF;
            {* end(transition) *}
            {* begin(onExit) *}
            {* end(onExit) *}
            {* end(State) *}

        Crane_states_t#No_Workpiece_ready:
            {* begin(State) *}
            {* begin(onEntry) *}
            _transit := FALSE;
            {* end(onEntry) *}
            {* begin(onActive) *}
            MagazinVacuumOn := FALSE;
            MagazinVacuumOff := FALSE;
            CraneLower := FALSE;
            {* end(onActive) *}
            {* begin(transition) *}
            IF StampSliderFilled THEN
                _transit := TRUE;
                _state := Crane_states_t#Crane_Turn_Left_Metallic2;
            ELSEIF NOT StampSliderFilled THEN
                _transit := TRUE;
                _state := Crane_states_t#Turn_Right_Final;
            END_IF;
            {* end(transition) *}
            {* begin(onExit) *}
            {* end(onExit) *}
            {* end(State) *}

        Crane_states_t#Reset_interconnect:
            {* begin(State) *}
            {* begin(onEntry) *}
            _transit := FALSE;
            {* end(onEntry) *}
            {* begin(onActive) *}
            interconnect := FALSE;
            Timer1(IN := FALSE, PT := TIME#1.0ms);
            {* end(onActive) *}
            {* begin(transition) *}
            IF SliderMovedOut THEN
                _transit := TRUE;
                _state := Crane_states_t#Lower_Crane;
            END_IF;
            {* end(transition) *}
            {* begin(onExit) *}
            {* end(onExit) *}
            {* end(State) *}

        Crane_states_t#Stamp_Pressure_Profile_Set_Metallic:
            {* begin(State) *}
            {* begin(onEntry) *}
            _transit := FALSE;
            {* end(onEntry) *}
            {* begin(onActive) *}
            AnalogCranePressure := INT#7000;
            {* end(onActive) *}
            {* begin(transition) *}
            IF TRUE THEN
                _transit := TRUE;
                _state := Crane_states_t#Crane_Lift_Magazin_Metallic;
            END_IF;
            {* end(transition) *}
            {* begin(onExit) *}
            {* end(onExit) *}
            {* end(State) *}

        Crane_states_t#Stamp_Pressure_Profile_Set_White:
            {* begin(State) *}
            {* begin(onEntry) *}
            _transit := FALSE;
            {* end(onEntry) *}
            {* begin(onActive) *}
            AnalogCranePressure := INT#6000;
            {* end(onActive) *}
            {* begin(transition) *}
            IF TRUE THEN
                _transit := TRUE;
                _state := Crane_states_t#Crane_Lift_Magazin_White;
            END_IF;
            {* end(transition) *}
            {* begin(onExit) *}
            {* end(onExit) *}
            {* end(State) *}

        Crane_states_t#Start_Crane:
            {* begin(State) *}
            {* begin(onEntry) *}
            _transit := FALSE;
            {* end(onEntry) *}
            {* begin(onActive) *}
            CraneLower := FALSE;
            MagazinVacuumOff := FALSE;
            MagazinVacuumOn := FALSE;
            CraneTurnCounterclockwise := FALSE;
            CraneTurnClockwise := FALSE;
            AnalogCranePressure := INT#0;
            StartVar := FALSE;
            StartCommandCrane := FALSE;
            IF (StartButtonMagazin = TRUE) THEN
                interconnectCraneStartCommand := TRUE;
            END_IF;
            {* end(onActive) *}
            {* begin(transition) *}
            IF interconnectCraneStartCommand THEN
                _transit := TRUE;
                _state := Crane_states_t#Crane_Init;
            END_IF;
            {* end(transition) *}
            {* begin(onExit) *}
            {* end(onExit) *}
            {* end(State) *}

        Crane_states_t#Step0:
            {* begin(State) *}
            {* begin(onEntry) *}
            _transit := FALSE;
            {* end(onEntry) *}
            {* begin(onActive) *}
            {* end(onActive) *}
            {* begin(transition) *}
            IF (MagazinCapacitiveSensor AND MagazinOpticalSensor) THEN
                _transit := TRUE;
                _state := Crane_states_t#Stamp_Pressure_Profile_Set_Metallic;
            ELSEIF (NOT MagazinCapacitiveSensor AND MagazinOpticalSensor) THEN
                _transit := TRUE;
                _state := Crane_states_t#Stamp_Pressure_Profile_Set_White;
            ELSEIF (NOT MagazinCapacitiveSensor AND NOT MagazinOpticalSensor) THEN
                _transit := TRUE;
                _state := Crane_states_t#Crane_Lift_Magazin;
            END_IF;
            {* end(transition) *}
            {* begin(onExit) *}
            {* end(onExit) *}
            {* end(State) *}

        Crane_states_t#Step2:
            {* begin(State) *}
            {* begin(onEntry) *}
            _transit := FALSE;
            {* end(onEntry) *}
            {* begin(onActive) *}
            {* end(onActive) *}
            {* begin(transition) *}
            IF (MagazinCapacitiveSensor OR MagazinOpticalSensor) THEN
                _transit := TRUE;
                _state := Crane_states_t#pause;
            ELSEIF (NOT MagazinCapacitiveSensor AND NOT MagazinOpticalSensor) THEN
                _transit := TRUE;
                _state := Crane_states_t#Turn_Right_Black;
            END_IF;
            {* end(transition) *}
            {* begin(onExit) *}
            {* end(onExit) *}
            {* end(State) *}

        Crane_states_t#Step3:
            {* begin(State) *}
            {* begin(onEntry) *}
            _transit := FALSE;
            {* end(onEntry) *}
            {* begin(onActive) *}
            {* end(onActive) *}
            {* begin(transition) *}
            IF NOT WorkpieceReady THEN
                _transit := TRUE;
                _state := Crane_states_t#Step4;
            ELSEIF WorkpieceReady THEN
                _transit := TRUE;
                _state := Crane_states_t#Step2;
            END_IF;
            {* end(transition) *}
            {* begin(onExit) *}
            {* end(onExit) *}
            {* end(State) *}

        Crane_states_t#Step4:
            {* begin(State) *}
            {* begin(onEntry) *}
            _transit := FALSE;
            {* end(onEntry) *}
            {* begin(onActive) *}
            {* end(onActive) *}
            {* begin(transition) *}
            IF TRUE THEN
                _transit := TRUE;
                _state := Crane_states_t#Interstep;
            END_IF;
            {* end(transition) *}
            {* begin(onExit) *}
            {* end(onExit) *}
            {* end(State) *}

        Crane_states_t#Suck_At_Stamp:
            {* begin(State) *}
            {* begin(onEntry) *}
            _transit := FALSE;
            {* end(onEntry) *}
            {* begin(onActive) *}
            MagazinVacuumOn := TRUE;
            MagazinVacuumOff := FALSE;
            {* end(onActive) *}
            {* begin(transition) *}
            IF CraneSucked THEN
                _transit := TRUE;
                _state := Crane_states_t#Crane_Lift_At_Stamp;
            END_IF;
            {* end(transition) *}
            {* begin(onExit) *}
            {* end(onExit) *}
            {* end(State) *}

        Crane_states_t#Suck_At_Stamp2:
            {* begin(State) *}
            {* begin(onEntry) *}
            _transit := FALSE;
            {* end(onEntry) *}
            {* begin(onActive) *}
            MagazinVacuumOn := TRUE;
            MagazinVacuumOff := FALSE;
            {* end(onActive) *}
            {* begin(transition) *}
            IF CraneSucked THEN
                _transit := TRUE;
                _state := Crane_states_t#Crane_Lift_At_Stamp2;
            END_IF;
            {* end(transition) *}
            {* begin(onExit) *}
            {* end(onExit) *}
            {* end(State) *}

        Crane_states_t#TimeDelay:
            {* begin(State) *}
            {* begin(onEntry) *}
            _transit := FALSE;
            {* end(onEntry) *}
            {* begin(onActive) *}
            TimeDelay_Timer(IN := TRUE, PT := TimeDelay_Timer_Duration);
            TimeDelay_Timer_interconnect := TimeDelay_Timer.Q;
            {* end(onActive) *}
            {* begin(transition) *}
            IF TimeDelay_Timer_interconnect THEN
                _transit := TRUE;
                _state := Crane_states_t#Interstep_3;
            END_IF;
            {* end(transition) *}
            {* begin(onExit) *}
            {* end(onExit) *}
            {* end(State) *}

        Crane_states_t#Turn_Right:
            {* begin(State) *}
            {* begin(onEntry) *}
            _transit := FALSE;
            {* end(onEntry) *}
            {* begin(onActive) *}
            CraneTurnClockwise := TRUE;
            CraneTurnCounterclockwise := FALSE;
            {* end(onActive) *}
            {* begin(transition) *}
            IF ((AnalogCranePosition > INT#24290) AND (AnalogCranePosition < INT#24390)) THEN
                _transit := TRUE;
                _state := Crane_states_t#Magazin_Stop;
            END_IF;
            {* end(transition) *}
            {* begin(onExit) *}
            {* end(onExit) *}
            {* end(State) *}

        Crane_states_t#Turn_Right_Black:
            {* begin(State) *}
            {* begin(onEntry) *}
            _transit := FALSE;
            {* end(onEntry) *}
            {* begin(onActive) *}
            CraneTurnClockwise := TRUE;
            CraneTurnCounterclockwise := FALSE;
            {* end(onActive) *}
            {* begin(transition) *}
            IF ((AnalogCranePosition > INT#24290) AND (AnalogCranePosition < INT#24390)) THEN
                _transit := TRUE;
                _state := Crane_states_t#Magazin_Stop_Black;
            END_IF;
            {* end(transition) *}
            {* begin(onExit) *}
            {* end(onExit) *}
            {* end(State) *}

        Crane_states_t#Turn_Right_Final:
            {* begin(State) *}
            {* begin(onEntry) *}
            _transit := FALSE;
            {* end(onEntry) *}
            {* begin(onActive) *}
            CraneTurnClockwise := TRUE;
            CraneTurnCounterclockwise := FALSE;
            AnalogCranePressure := INT#0;
            {* end(onActive) *}
            {* begin(transition) *}
            IF ((AnalogCranePosition > INT#24290) AND (AnalogCranePosition < INT#24390)) THEN
                _transit := TRUE;
                _state := Crane_states_t#Magazin_Stop_Final;
            END_IF;
            {* end(transition) *}
            {* begin(onExit) *}
            {* end(onExit) *}
            {* end(State) *}

        Crane_states_t#pause:
            {* begin(State) *}
            {* begin(onEntry) *}
            _transit := FALSE;
            {* end(onEntry) *}
            {* begin(onActive) *}
            Timer1(IN := CraneUp, PT := Duration1);
            interconnect := Timer1.Q;
            {* end(onActive) *}
            {* begin(transition) *}
            IF interconnect THEN
                _transit := TRUE;
                _state := Crane_states_t#Reset_interconnect;
            END_IF;
            {* end(transition) *}
            {* begin(onExit) *}
            {* end(onExit) *}
            {* end(State) *}

        Crane_states_t#release:
            {* begin(State) *}
            {* begin(onEntry) *}
            _transit := FALSE;
            {* end(onEntry) *}
            {* begin(onActive) *}
            MagazinVacuumOff := TRUE;
            MagazinVacuumOn := FALSE;
            {* end(onActive) *}
            {* begin(transition) *}
            IF TRUE THEN
                _transit := TRUE;
                _state := Crane_states_t#Crane_Lift_Conveyor;
            END_IF;
            {* end(transition) *}
            {* begin(onExit) *}
            {* end(onExit) *}
            {* end(State) *}

        Crane_states_t#release2:
            {* begin(State) *}
            {* begin(onEntry) *}
            _transit := FALSE;
            {* end(onEntry) *}
            {* begin(onActive) *}
            MagazinVacuumOff := TRUE;
            MagazinVacuumOn := FALSE;
            {* end(onActive) *}
            {* begin(transition) *}
            IF TRUE THEN
                _transit := TRUE;
                _state := Crane_states_t#Crane_Lift_Conveyor2;
            END_IF;
            {* end(transition) *}
            {* begin(onExit) *}
            {* end(onExit) *}
            {* end(State) *}

        Crane_states_t#release_Black:
            {* begin(State) *}
            {* begin(onEntry) *}
            _transit := FALSE;
            {* end(onEntry) *}
            {* begin(onActive) *}
            MagazinVacuumOn := FALSE;
            MagazinVacuumOff := TRUE;
            {* end(onActive) *}
            {* begin(transition) *}
            IF TRUE THEN
                _transit := TRUE;
                _state := Crane_states_t#Crane_Lift_Conveyor_Black;
            END_IF;
            {* end(transition) *}
            {* begin(onExit) *}
            {* end(onExit) *}
            {* end(State) *}

        Crane_states_t#release_Workpiece:
            {* begin(State) *}
            {* begin(onEntry) *}
            _transit := FALSE;
            {* end(onEntry) *}
            {* begin(onActive) *}
            MagazinVacuumOff := TRUE;
            MagazinVacuumOn := FALSE;
            {* end(onActive) *}
            {* begin(transition) *}
            IF TRUE THEN
                _transit := TRUE;
                _state := Crane_states_t#Crane_Go_Up;
            END_IF;
            {* end(transition) *}
            {* begin(onExit) *}
            {* end(onExit) *}
            {* end(State) *}

        Crane_states_t#release_Workpiece_White:
            {* begin(State) *}
            {* begin(onEntry) *}
            _transit := FALSE;
            {* end(onEntry) *}
            {* begin(onActive) *}
            MagazinVacuumOff := TRUE;
            MagazinVacuumOn := FALSE;
            {* end(onActive) *}
            {* begin(transition) *}
            IF TRUE THEN
                _transit := TRUE;
                _state := Crane_states_t#Crane_Go_Up_White;
            END_IF;
            {* end(transition) *}
            {* begin(onExit) *}
            {* end(onExit) *}
            {* end(State) *}

            END_CASE;
END_FUNCTION_BLOCK

(* ---- Scenario13_Final.xml_Magazin.st ---- *)
FUNCTION_BLOCK Magazin
    VAR_INPUT  AnalogCranePosition : INT; END_VAR {*Irwxp*}
    VAR_INPUT  CraneDown : BOOL; END_VAR {*Irwxp*}
    VAR_OUTPUT  CraneLower : BOOL; END_VAR {*Orwxp*}
    VAR_INPUT  CraneOnConveyor : BOOL; END_VAR {*Irwxp*}
    VAR_INPUT  CraneOnMagazin : BOOL; END_VAR {*Irwxp*}
    VAR_INPUT  CraneSucked : BOOL; END_VAR {*Irwxp*}
    VAR_OUTPUT  CraneTurnClockwise : BOOL; END_VAR {*Orwxp*}
    VAR_OUTPUT  CraneTurnCounterclockwise : BOOL; END_VAR {*Orwxp*}
    VAR_INPUT  CraneUp : BOOL; END_VAR {*Irwxp*}
    VAR_OUTPUT  MagazinGreenLamp : BOOL; END_VAR {*Orwxp*}
    VAR_OUTPUT  MagazinSlider : BOOL; END_VAR {*Orwxp*}
    VAR_OUTPUT  MagazinVacuumOff : BOOL; END_VAR {*Orwxp*}
    VAR_OUTPUT  MagazinVacuumOn : BOOL; END_VAR {*Orwxp*}
    VAR_OUTPUT  MagazinWhiteLamp : BOOL; END_VAR {*Orwxp*}
    VAR  SFCInit : BOOL; END_VAR {*Lrwxp*}
    VAR_INPUT  SFCReset : BOOL; END_VAR {*Irwxp*}
    VAR_INPUT  SliderMovedOut : BOOL; END_VAR {*Irwxp*}
    VAR_INPUT  SliderNotMovedOut : BOOL; END_VAR {*Irwxp*}
    VAR_INPUT  StartButtonMagazin : BOOL; END_VAR {*Irwxp*}
    VAR_OUTPUT  StartCommandMagazin : BOOL; END_VAR {*Orwxp*}
    VAR_INPUT  StartVar : BOOL; END_VAR {*Irwxp*}
    VAR_INPUT  WorkpieceReady : BOOL; END_VAR {*Irwxp*}
    VAR  _state : Magazin_states_t; END_VAR {*Lrwxp*}
    VAR  _transit : BOOL; END_VAR {*Lrwxp*}
    VAR  interconnectMagazinStartCommand : BOOL; END_VAR {*Lrwxp*}

    CASE _state OF
        Magazin_states_t#Green_Lamp:
            {* begin(State) *}
            {* begin(onEntry) *}
            _transit := FALSE;
            {* end(onEntry) *}
            {* begin(onActive) *}
            MagazinGreenLamp := TRUE;
            interconnectMagazinStartCommand := FALSE;
            {* end(onActive) *}
            {* begin(transition) *}
            IF TRUE THEN
                _transit := TRUE;
                _state := Magazin_states_t#Magazin_Init;
            END_IF;
            {* end(transition) *}
            {* begin(onExit) *}
            {* end(onExit) *}
            {* end(State) *}

        Magazin_states_t#Init:
            {* begin(State) *}
            {* begin(onEntry) *}
            _transit := FALSE;
            {* end(onEntry) *}
            {* begin(onActive) *}
            {* end(onActive) *}
            {* begin(transition) *}
            IF TRUE THEN
                _transit := TRUE;
                _state := Magazin_states_t#Start_Magazin;
            END_IF;
            {* end(transition) *}
            {* begin(onExit) *}
            {* end(onExit) *}
            {* end(State) *}

        Magazin_states_t#Interstep:
            {* begin(State) *}
            {* begin(onEntry) *}
            _transit := FALSE;
            {* end(onEntry) *}
            {* begin(onActive) *}
            StartCommandMagazin := TRUE;
            {* end(onActive) *}
            {* begin(transition) *}
            IF StartVar THEN
                _transit := TRUE;
                _state := Magazin_states_t#convey;
            END_IF;
            {* end(transition) *}
            {* begin(onExit) *}
            {* end(onExit) *}
            {* end(State) *}

        Magazin_states_t#Magazin_Init:
            {* begin(State) *}
            {* begin(onEntry) *}
            _transit := FALSE;
            {* end(onEntry) *}
            {* begin(onActive) *}
            MagazinSlider := TRUE;
            {* end(onActive) *}
            {* begin(transition) *}
            IF TRUE THEN
                _transit := TRUE;
                _state := Magazin_states_t#Magazin_Init_2;
            END_IF;
            {* end(transition) *}
            {* begin(onExit) *}
            {* end(onExit) *}
            {* end(State) *}

        Magazin_states_t#Magazin_Init_2:
            {* begin(State) *}
            {* begin(onEntry) *}
            _transit := FALSE;
            {* end(onEntry) *}
            {* begin(onActive) *}
            MagazinSlider := FALSE;
            {* end(onActive) *}
            {* begin(transition) *}
            IF TRUE THEN
                _transit := TRUE;
                _state := Magazin_states_t#Interstep;
            END_IF;
            {* end(transition) *}
            {* begin(onExit) *}
            {* end(onExit) *}
            {* end(State) *}

        Magazin_states_t#Slider_Move_Back:
            {* begin(State) *}
            {* begin(onEntry) *}
            _transit := FALSE;
            {* end(onEntry) *}
            {* begin(onActive) *}
            IF ((SliderMovedOut = TRUE) AND (SliderNotMovedOut = FALSE)) THEN
                MagazinSlider := FALSE;
            END_IF;
            {* end(onActive) *}
            {* begin(transition) *}
            IF CraneUp THEN
                _transit := TRUE;
                _state := Magazin_states_t#Step1;
            END_IF;
            {* end(transition) *}
            {* begin(onExit) *}
            {* end(onExit) *}
            {* end(State) *}

        Magazin_states_t#Start_Magazin:
            {* begin(State) *}
            {* begin(onEntry) *}
            _transit := FALSE;
            {* end(onEntry) *}
            {* begin(onActive) *}
            MagazinSlider := FALSE;
            MagazinGreenLamp := FALSE;
            StartVar := FALSE;
            StartCommandMagazin := FALSE;
            IF (StartButtonMagazin = TRUE) THEN
                interconnectMagazinStartCommand := TRUE;
            END_IF;
            {* end(onActive) *}
            {* begin(transition) *}
            IF interconnectMagazinStartCommand THEN
                _transit := TRUE;
                _state := Magazin_states_t#Green_Lamp;
            END_IF;
            {* end(transition) *}
            {* begin(onExit) *}
            {* end(onExit) *}
            {* end(State) *}

        Magazin_states_t#Step0:
            {* begin(State) *}
            {* begin(onEntry) *}
            _transit := FALSE;
            {* end(onEntry) *}
            {* begin(onActive) *}
            {* end(onActive) *}
            {* begin(transition) *}
            IF CraneDown THEN
                _transit := TRUE;
                _state := Magazin_states_t#Slider_Move_Back;
            END_IF;
            {* end(transition) *}
            {* begin(onExit) *}
            {* end(onExit) *}
            {* end(State) *}

        Magazin_states_t#Step1:
            {* begin(State) *}
            {* begin(onEntry) *}
            _transit := FALSE;
            {* end(onEntry) *}
            {* begin(onActive) *}
            {* end(onActive) *}
            {* begin(transition) *}
            IF ((AnalogCranePosition > INT#16160) AND (AnalogCranePosition < INT#16260)) THEN
                _transit := TRUE;
                _state := Magazin_states_t#Interstep;
            END_IF;
            {* end(transition) *}
            {* begin(onExit) *}
            {* end(onExit) *}
            {* end(State) *}

        Magazin_states_t#convey:
            {* begin(State) *}
            {* begin(onEntry) *}
            _transit := FALSE;
            {* end(onEntry) *}
            {* begin(onActive) *}
            IF SliderNotMovedOut THEN
                MagazinSlider := TRUE;
            END_IF;
            {* end(onActive) *}
            {* begin(transition) *}
            IF ((AnalogCranePosition > INT#24290) AND (AnalogCranePosition < INT#24390)) THEN
                _transit := TRUE;
                _state := Magazin_states_t#Step0;
            END_IF;
            {* end(transition) *}
            {* begin(onExit) *}
            {* end(onExit) *}
            {* end(State) *}

            END_CASE;
END_FUNCTION_BLOCK
